// TIA Portal V20 export
DATA_BLOCK "SqlConfig"   // DB7
TITLE = SqlConfig
{ S7_Optimized_Access := 'TRUE' }
AUTHOR : SIEMENS SUP Applications
VERSION : 1.1
// DB for providing the connection settings for a Tabuar Data Stream to a SQL database
// stored: MemoryReserve 100
   VAR
      connectionSettings { ExternalAccessible := 'False'; ExternalVisible := 'False'; ExternalWritable := 'False'} : "LSql_typeConnectionSettings";
      enableLSql { ExternalAccessible := 'False'; ExternalVisible := 'False'; ExternalWritable := 'False'} : Bool;   // enables LSql block (starts connection and login, waits for execute commands)
      diagnostics { ExternalWritable := 'False'} : "LSql_typeDiagnostics";
      executeSqlCommand { ExternalAccessible := 'False'; ExternalVisible := 'False'; ExternalWritable := 'False'} : Bool;   // trigger to execute a single sql command. EnableLSql must be true before triggering
   END_VAR
BEGIN
   connectionSettings.interfaceSettings.InterfaceId := 64;
   connectionSettings.interfaceSettings.ID := 16#10;
   connectionSettings.interfaceSettings.ActiveEstablished := true;
   connectionSettings.interfaceSettings.RemoteAddress.ADDR[1] := 10;
   connectionSettings.interfaceSettings.RemoteAddress.ADDR[2..3] := 30;
   connectionSettings.interfaceSettings.RemoteAddress.ADDR[4] := 222;
   connectionSettings.interfaceSettings.RemotePort := 1433;
   connectionSettings.loginInformation.userName := 'SQL_S71500';
   connectionSettings.loginInformation.password := 'SQL_S71500';
   connectionSettings.loginInformation.serverName := 'SQLEXPRESS';
   connectionSettings.loginInformation.databaseName := 'S71500SQLDB';
END_DATA_BLOCK
